{attribute 'GeneratedUsingTerminal: EK1100-0000-0018'}
{attribute addProperty BoxType "EK1100-0000-0018"}
{attribute addProperty Id "Beckhoff_ELM9xxxEK1122Beckhoff_ELM9xxxEK1122_C85844232A_0002_ELM9410_0000_0016ELM9410_DD55393581A_0003_ELM9410_0000_0017ELM9410_DD55393581A_0004_ELM9410_0000_0018ELM9410_DD55393581A_0005_ELM9410_0000_0019ELM9410_DD55393581A_0006_ELM9410_0000_0020ELM9410_DD55393581"}
{attribute addProperty CRC "980777355"}
{attribute addProperty Size "407"}
TYPE Beckhoff_ELM9xxx_3A75798B EXTENDS EK1100_1FC0878B :
STRUCT
	{attribute addProperty Name "Beckhoff_ELM9xxxEK1122"}
	Beckhoff_ELM9xxxEK1122 : Beckhoff_ELM9xxxEK1122_C8584423;
	{attribute addProperty Name "A_0002_ELM9410_0000_0016"}
	A_0002_ELM9410_0000_0016 : ELM9410_DD553935;
	{attribute addProperty Name "A_0003_ELM9410_0000_0017"}
	A_0003_ELM9410_0000_0017 : ELM9410_DD553935;
	{attribute addProperty Name "A_0004_ELM9410_0000_0018"}
	A_0004_ELM9410_0000_0018 : ELM9410_DD553935;
	{attribute addProperty Name "A_0005_ELM9410_0000_0019"}
	A_0005_ELM9410_0000_0019 : ELM9410_DD553935;
	{attribute addProperty Name "A_0006_ELM9410_0000_0020"}
	A_0006_ELM9410_0000_0020 : ELM9410_DD553935;
END_STRUCT
END_TYPE

(* stored: Version 1.2.0.0, ProductVersion 3.1.4024.9
   DUT Beckhoff_ELM9xxx_3A75798B: Id {90f0a388-e406-4b16-9e38-1212e27ff934} *)
